FUNCTION_BLOCK SimulationFB
VAR_IN_OUT
	Parameters: GreenMasterBaseParameters;
END_VAR
VAR_INPUT
	Simulation: SimulationParameters;	
END_VAR
VAR_OUTPUT
END_VAR
VAR
END_VAR

Main.GreenMaster.Simulate(Parameters := Main.GreenMaster.GetParameters(),
	ParametersFB := Main.GreenMaster.GetParametersFB());

END_FUNCTION_BLOCK

(* stored: Version 1.1.0.1, ProductVersion 3.1.4024.6
   POU SimulationFB: Id {e07fe9b8-b0ad-45ff-a31d-c7901da29d36}, SpecialFunc None *)
